(* IEC 61131-3 sources: generating_plc_code_with_llms/Code#1/ChatGPT_3.5/first run, 20 files *)

(* ---- 10.st ---- *)
//7.60s
//2
FUNCTION Sigmoid : REAL
VAR_INPUT
    x: REAL;  // Input value for the sigmoid function
END_VAR_INPUT
VAR_OUTPUT
    result: REAL;  // Result of the sigmoid function
END_VAR_OUTPUT

VAR
    exp_neg_x: REAL;
BEGIN
    exp_neg_x := EXP(-x);
    result := 1 / (1 + exp_neg_x);
END_FUNCTION

(* ---- 11.st ---- *)
//7.59s
//2
FUNCTION Sign : INT
VAR_INPUT
    value: REAL;  // Input value to determine the sign of
END_VAR_INPUT
VAR_OUTPUT
    sign: INT;    // Output sign value (-1, 0, or 1)
END_VAR_OUTPUT
BEGIN
    IF value < 0 THEN
        sign := -1;
    ELSIF value = 0 THEN
        sign := 0;
    ELSE
        sign := 1;
    END_IF
END_FUNCTION

(* ---- 12.st ---- *)
//8.05s
//2
FUNCTION HyperbolicSine : REAL
VAR_INPUT
    x: REAL;  // Input value for the hyperbolic sine function
END_VAR_INPUT
VAR_OUTPUT
    result: REAL;  // Result of the hyperbolic sine function
END_VAR_OUTPUT

VAR
    exp_x: REAL;
    exp_neg_x: REAL;
BEGIN
    exp_x := EXP(x);
    exp_neg_x := EXP(-x);
    result := (exp_x - exp_neg_x) / 2;
END_FUNCTION

(* ---- 14.st ---- *)
// 33.60s
// 3
FUNCTION FC1001 : BOOL
VAR_INPUT
    MeasuredValue: REAL;      // Measured value from the sensor
    SwitchingValue: REAL;     // Predetermined switching value
    HysteresisPercent: REAL;  // Switching hysteresis in percentage
END_VAR

VAR_OUTPUT
    Output: BOOL;  // Output indicating the state (ON or OFF)
END_VAR

VAR
    HysteresisValue: REAL;  // Calculated hysteresis value based on percentage
    SwitchOnThreshold: REAL; // Threshold for switching ON
    SwitchOffThreshold: REAL; // Threshold for switching OFF
END_VAR

METHOD CheckSwitching
    HysteresisValue := SwitchingValue * HysteresisPercent / 100.0;

    SwitchOnThreshold := SwitchingValue + HysteresisValue;
    SwitchOffThreshold := SwitchingValue - HysteresisValue;

    IF MeasuredValue > SwitchOnThreshold THEN
        Output := TRUE;  // Switch ON
    ELSIF MeasuredValue < SwitchOffThreshold THEN
        Output := FALSE; // Switch OFF
    END_IF
END_METHOD

END_FUNCTION

(* ---- 15.st ---- *)
// 25.63s
// 2
FUNCTION FC1002 : BOOL
VAR_INPUT
    E_A: BOOL;    // Switch for turning on/off the monitoring system
    Approach: BOOL;  // Signal from the ultrasonic sensor indicating an approach
END_VAR

VAR_OUTPUT
    P_HU: BOOL;  // Output for the acoustic warning signal
    P_AL: BOOL;  // Output for the alarm signal
    P1: BOOL;    // Output indicating the switched-on status
END_VAR

VAR
    Timer: TON := (PT := T#3s);  // Timer for tracking the duration of the approach
END_VAR

METHOD UltrasonicMonitoring
    IF E_A THEN
        P1 := TRUE;  // Monitoring system is switched on

        IF Approach THEN
            P_HU := TRUE;  // Acoustic warning signal is activated

            IF Timer(IN := TRUE).Q THEN
                // Approach duration exceeds 3 seconds, switch off warning and activate alarm
                P_HU := FALSE;
                P_AL := TRUE;
            END_IF
        ELSE
            // No approach, reset the timer and signals
            Timer(IN := FALSE);
            P_HU := FALSE;
            P_AL := FALSE;
        END_IF
    ELSE
        // Monitoring system is switched off, reset all signals
        P1 := FALSE;
        P_HU := FALSE;
        P_AL := FALSE;
        Timer(IN := FALSE);
    END_IF
END_METHOD

END_FUNCTION

(* ---- 18.st ---- *)
// 8.55s
// 2
FUNCTION FC1003
VAR_INPUT
    DigitalInput: INT;  // Digital input value (0 to 255)
    IN_MIN: INT;        // Lower limit of the original range
    IN_MAX: INT;        // Upper limit of the original range
    OUT_MIN: REAL;      // Lower limit of the output range
    OUT_MAX: REAL;      // Upper limit of the output range
END_VAR_INPUT

VAR_OUTPUT
    Temperature: REAL;  // Converted temperature value
END_VAR_OUTPUT

VAR
    M: REAL;            // Slope of the linear mapping
    B: REAL;            // Y-intercept of the linear mapping
END_VAR

// Calculate the slope and y-intercept for the linear mapping
M := (OUT_MAX - OUT_MIN) / (IN_MAX - IN_MIN);
B := OUT_MIN - M * IN_MIN;

// Perform the linear mapping to convert DigitalInput to Temperature
Temperature := M * DigitalInput + B;

END_FUNCTION

(* ---- 2.st ---- *)
//7.4s
//2
FUNCTION CalculateBinomialCoefficient : INT
VAR_INPUT
    n : INT;  // The total number of items (n)
    k : INT;  // The number of items to choose (k)
END_VAR_INPUT
VAR_OUTPUT
    result : INT;  // The binomial coefficient result
END_VAR_OUTPUT
VAR
    i : INT;
    numerator : INT := 1;
    denominator : INT := 1;
END_VAR

IF (k < 0) OR (k > n) THEN
    result := 0;  // Invalid input, return 0
ELSE
    FOR i := 1 TO k DO
        numerator := numerator * (n - i + 1);
        denominator := denominator * i;
    END_FOR

    result := numerator / denominator;
END_IF

END_FUNCTION

(* ---- 3.st ---- *)
//6.85s
//2
FUNCTION CalculateFibonacci : INT
VAR_INPUT
    n : INT;  // The position in the Fibonacci sequence (0-based)
END_VAR_INPUT
VAR_OUTPUT
    result : INT;  // The Fibonacci number at position 'n'
END_VAR_OUTPUT
VAR
    fibNMinus2 : INT := 0;  // Initial values for the first two Fibonacci numbers
    fibNMinus1 : INT := 1;
    fibN : INT;
    i : INT;
END_VAR

IF n = 0 THEN
    result := fibNMinus2;  // Special case for n = 0
ELSIF n = 1 THEN
    result := fibNMinus1;  // Special case for n = 1
ELSE
    FOR i := 2 TO n DO
        fibN := fibNMinus1 + fibNMinus2;
        fibNMinus2 := fibNMinus1;
        fibNMinus1 := fibN;
    END_FOR

    result := fibN;
END_IF

END_FUNCTION

(* ---- 19.st ---- *)
// 20.66s
// 3
FUNCTION_BLOCK FB1005
VAR_INPUT
    START: BOOL;      // Start the measurement (connected to sensor S1)
    THICKNESS: REAL;  // Input representing the thickness of the ceramic plate
    V_MAX: REAL;      // Maximum allowed thickness
    V_MIN: REAL;      // Minimum allowed thickness
END_VAR

VAR_OUTPUT
    M_MAX: REAL;      // Largest thickness recorded during the measurement
    M_MIN: REAL;      // Smallest thickness recorded during the measurement
    P1: BOOL;         // Output for the reject light
END_VAR

VAR
    D_MAX: BOOL;      // Flag indicating if the largest thickness is outside the specified range
    D_MIN: BOOL;      // Flag indicating if the smallest thickness is outside the specified range
    ThicknessStarted: BOOL;  // Flag indicating if the thickness measurement has started
    LastThickness: REAL;     // Last recorded thickness during the measurement
END_VAR

METHOD MeasureThickness
    IF START THEN
        // Start of a new measurement cycle
        M_MAX := THICKNESS;  // Initialize largest thickness
        M_MIN := THICKNESS;  // Initialize smallest thickness
        D_MAX := FALSE;      // Initialize flags
        D_MIN := FALSE;
        ThicknessStarted := TRUE;  // Set the flag to indicate the measurement has started
    END_IF

    IF ThicknessStarted THEN
        // During the measurement cycle
        IF THICKNESS > M_MAX THEN
            M_MAX := THICKNESS;  // Update largest thickness
        END_IF

        IF THICKNESS < M_MIN THEN
            M_MIN := THICKNESS;  // Update smallest thickness
        END_IF

        LastThickness := THICKNESS;  // Record the last thickness
    END_IF

    // After the measurement cycle
    IF NOT START AND ThicknessStarted THEN
        ThicknessStarted := FALSE;  // Reset the flag to indicate the end of the measurement
        D_MAX := M_MAX > V_MAX;     // Check if the largest thickness is outside the specified range
        D_MIN := M_MIN < V_MIN;     // Check if the smallest thickness is outside the specified range
    END_IF

    // Output the reject light signal
    P1 := D_MAX OR D_MIN;
END_METHOD

END_FUNCTION_BLOCK

(* ---- 21.st ---- *)
// 46.74s
// 2
FUNCTION_BLOCK BURNER
VAR_INPUT
    IN: BOOL;                  // Control input
    OVER_TEMP: BOOL;           // Boiler thermostat protection
    OIL_TEMP: BOOL;            // Signal indicating oil temperature reached
    MULTIPLE_IGNITION: BOOL;   // Enable multiple ignition after flame break
    STAGE2: BOOL;              // Activate second stage
END_VAR_INPUT

VAR_OUTPUT
    PRE_HEAT: BOOL;            // Fuel oil warming
    MOTOR: BOOL;               // Motor status
    FAN: BOOL;                 // Fan status
    IGNITION: BOOL;            // Ignition status
    OIL_VALVE: BOOL;           // Oil valve status
    STATUS: INT;               // Module status
    FAIL: BOOL;                // Failure indication
END_VAR_OUTPUT

VAR
    startTime: TIME;           // Start time for various stages
    locked: BOOL;              // Module lock status
END_VAR

METHOD StartBurner : BOOL
VAR
    elapsedTime: TIME;         // Elapsed time for various stages
BEGIN
    // Check if the module is locked
    IF locked THEN
        STATUS := 99;  // Module is locked
        RETURN FALSE;
    END_IF

    // Reset failure indication
    FAIL := FALSE;

    // Start sequence
    IF IN AND NOT OVER_TEMP THEN
        PRE_HEAT := TRUE;  // Fuel oil warming
        startTime := T;    // Record start time

        // Wait for OIL_TEMP signal within PRE_HEAT_TIME
        WHILE (T - startTime < PRE_HEAT_TIME) AND NOT OIL_TEMP DO
            // Check if OVER_TEMP signal received during waiting
            IF OVER_TEMP THEN
                STATUS := 9;  // Boiler overheating error
                RETURN FALSE;
            END_IF
        END_WHILE

        // Check if OIL_TEMP signal received within PRE_HEAT_TIME
        IF OIL_TEMP THEN
            MOTOR := TRUE;  // Start motor
            FAN := TRUE;    // Start fan

            // Wait for PRE_VENTILATION_TIME before ignition
            WHILE (T - startTime < PRE_VENTILATION_TIME) DO
                // Check if OVER_TEMP signal received during waiting
                IF OVER_TEMP THEN
                    STATUS := 9;  // Boiler overheating error
                    RETURN FALSE;
                END_IF
            END_WHILE

            IGNITION := TRUE;  // Turn on ignition

            // Wait for PPR_IGNITION_TIME before opening oil valve
            WHILE (T - startTime < PPR_IGNITION_TIME) DO
                // Check if OVER_TEMP signal received during waiting
                IF OVER_TEMP THEN
                    STATUS := 9;  // Boiler overheating error
                    RETURN FALSE;
                END_IF
            END_WHILE

            OIL_VALVE := TRUE;  // Open oil valve

            // Wait for POST_IGNITION_TIME after ignition
            WHILE (T - startTime < POST_IGNITION_TIME) DO
                // Check if OVER_TEMP signal received during waiting
                IF OVER_TEMP THEN
                    STATUS := 9;  // Boiler overheating error
                    RETURN FALSE;
                END_IF
            END_WHILE

            // Check if flame sensor is active during SAFETY_TIME
            IF FLAME_SENSOR_ACTIVE(DURATION := SAFETY_TIME) THEN
                STATUS := 4;  // Safety time error
                RETURN FALSE;
            END_IF

            // Successful operation in stage 1
            STATUS := 112;  // Burner runs on stage 1

            // If MULTIPLE_IGNITION is enabled and flame breaks off, restart ignition
            IF MULTIPLE_IGNITION AND FLAME_SENSOR_ACTIVE(DURATION := MULTIPLE_IGNITION_TIME) THEN
                IGNITION := TRUE;  // Restart ignition
            END_IF

            // Check if second stage is activated
            IF STAGE2 THEN
                // Wait for STAGE2_DELAY before activating second stage
                WHILE (T - startTime < STAGE2_DELAY) DO
                    // Check if OVER_TEMP signal received during waiting
                    IF OVER_TEMP THEN
                        STATUS := 9;  // Boiler overheating error
                        RETURN FALSE;
                    END_IF
                END_WHILE

                // Activate second stage
                STATUS := 113;  // Burner runs at stage 2
            END_IF

            // Burner operation completed successfully
            RETURN TRUE;
        ELSE
            // OIL_TEMP signal not received within PRE_HEAT_TIME
            STATUS := 1;  // Fuel oil warming not responded error
            FAIL := TRUE;
            RETURN FALSE;
        END_IF
    ELSE
        // IN or OVER_TEMP condition not met
        STATUS := 110;  // Wait for Start signal (Standby)
        RETURN FALSE;
    END_IF
END_METHOD

METHOD FLAME_SENSOR_ACTIVE : BOOL
VAR_INPUT
    DURATION: TIME;  // Duration to check flame sensor activity
END_VAR_INPUT

VAR
    startTime: TIME;  // Start time for flame sensor check
BEGIN
    startTime := T;

    WHILE (T - startTime < DURATION) DO
        // Check if flame sensor is active
        IF FLAME_SENSOR THEN
            STATUS := 2;  // Flame sensor active error
            FAIL := TRUE;
            RETURN TRUE;
        END_IF
    END_WHILE

    // Flame sensor not active within specified duration
    RETURN FALSE;
END_METHOD

METHOD Lockout : BOOL
VAR
    lockoutStartTime: TIME;  // Start time for lockout
BEGIN
    // Set the module to locked state
    locked := TRUE;

    // Start lockout timer
    lockoutStartTime := T;

    // Wait for LOCKOUT_TIME
    WHILE (T - lockoutStartTime < LOCKOUT_TIME) AND NOT RST DO
        // Check if OVER_TEMP signal received during waiting
        IF OVER_TEMP THEN
            STATUS := 9;  // Boiler overheating error
            FAIL := TRUE;
            RETURN FALSE;
        END_IF
    END_WHILE

    // Reset the module lock
    locked := FALSE;

    // Module is ready for operation again
    STATUS := 110;  // Wait for Start signal (Standby)

    // Return TRUE if RST signal received after LOCKOUT_TIME
    RETURN RST;
END_METHOD

END_FUNCTION_BLOCK

(* ---- 1.st ---- *)
// 5.73s
//3
PROGRAM AlarmControl
VAR
    xAlarm1: BOOL := FALSE;
    xAlarm2: BOOL := FALSE;
    xAllOn: BOOL := FALSE;
    xAllOff: BOOL := FALSE;
END_VAR

xAlarm1 := FALSE;  // Ensure alarms are initially turned off
xAlarm2 := FALSE;

IF xAllOn THEN
    xAlarm1 := TRUE;
    xAlarm2 := TRUE;
ELSIF xAllOff THEN
    xAlarm1 := FALSE;
    xAlarm2 := FALSE;
END_IF

// Rest of your program logic here

END_PROGRAM

(* ---- 13.st ---- *)
//12.85s
//2
PROGRAM NumberSearch
VAR
    NumberList: ARRAY[1..100] OF INT;  // Array of 100 random numbers
    NumberToFind: INT := 10;           // Number to search for
    NumberFound: BOOL := FALSE;        // Flag to indicate if the number is found
    i: INT := 1;                       // Loop counter
END_VAR

FOR i := 1 TO 100 DO
    NumberList[i] := RANDOM(1, 100);  // Replace with a function that generates random numbers

    IF NumberList[i] = NumberToFind THEN
        NumberFound := TRUE;  // The number 10 is found, abort the search
        EXIT;  // Exit the loop
    END_IF
END_FOR

IF NOT NumberFound THEN
    // The number 10 was not found in the list
    // Handle the case where the number does not exist
    // Your logic for this case goes here
END_IF

// Your program logic continues here

(* ---- 16.st ---- *)
//13.22s
//2
PROGRAM TrafficLightControl
VAR
    North_green: BOOL := FALSE;
    North_yellow: BOOL := FALSE;
    North_red: BOOL := FALSE;
    East_green: BOOL := FALSE;
    East_yellow: BOOL := FALSE;
    East_red: BOOL := FALSE;

    TrafficLightCycleTimer: TON := (PT := T#10000ms);
END_VAR

CASE TrafficLightCycleTimer.IN THEN
    0:  // Between 0ms and 5000ms
        North_green := TRUE;
        East_green := FALSE;
        East_red := TRUE;
    5000:  // After 5000ms, North light turns yellow
        North_green := FALSE;
        North_yellow := TRUE;
    5500:  // Between 5500ms and 9500ms
        North_yellow := FALSE;
        North_red := TRUE;
        East_green := TRUE;
        East_red := FALSE;
    9500:  // Between 9500ms and 10000ms
        East_green := FALSE;
        East_yellow := TRUE;
    10000:  // Reset the timer and the cycle
        TrafficLightCycleTimer(IN := FALSE, PT := T#10000ms);
        North_red := FALSE;
        East_yellow := FALSE;
        North_green := TRUE;
        East_red := TRUE;
END_CASE

TrafficLightCycleTimer(IN := TRUE);

(* ---- 17.st ---- *)
//10.91s
//4
PROGRAM WeatherStation
VAR
    TemperatureSensorValue: INT;   // Analog input value for temperature
    HumiditySensorValue: INT;      // Analog input value for humidity
    TemperatureText: STRING := ''; // Text representation of temperature status
    HumidityText: STRING := '';    // Text representation of humidity status
END_VAR

TemperatureSensorValue := YourTemperatureSensorFunction(); // Replace with your sensor reading
HumiditySensorValue := YourHumiditySensorFunction();       // Replace with your sensor reading

IF TemperatureSensorValue < 18 THEN
    TemperatureText := 'Cold';
ELSIF TemperatureSensorValue >= 18 AND TemperatureSensorValue <= 25 THEN
    IF HumiditySensorValue >= 40 AND HumiditySensorValue <= 75 THEN
        TemperatureText := 'Opt';
    ELSE
        TemperatureText := 'Temp. OK';
    END_IF;
ELSE
    TemperatureText := 'Hot';
END_IF

// Display the temperature status in the house
DISPLAY_IN_HOUSE(TemperatureText);

// Your program logic continues here

END_PROGRAM

(* ---- 20.st ---- *)
// 15.67s
// 3
PROGRAM InterlockProgram
VAR_INPUT
    I1: BOOL;  // Input to switch Q1
    I2: BOOL;  // Input to switch Q2
END_VAR

VAR_OUTPUT
    Q1: BOOL;  // Output Q1
    Q2: BOOL;  // Output Q2
END_VAR

VAR
    TimerQ1: TON := (PT := T#1s);  // Timer for Q1
    TimerQ2: TON := (PT := T#1s);  // Timer for Q2
    TL: TIME := T#500ms;           // Dead time between Q1 and Q2
    LastQ1State: BOOL := FALSE;    // Last state of Q1
    LastQ2State: BOOL := FALSE;    // Last state of Q2
END_VAR

METHOD InterlockLogic
    // Update timers
    TimerQ1(IN := I1);
    TimerQ2(IN := I2);

    // Determine the next state of Q1
    IF I1 AND NOT Q2 AND TimerQ2.Q THEN
        Q1 := TRUE;
        LastQ1State := TRUE;
    ELSIF NOT I1 THEN
        Q1 := FALSE;
        TimerQ1(IN := FALSE);  // Reset the timer if I1 is OFF
    END_IF

    // Determine the next state of Q2
    IF I2 AND NOT Q1 AND TimerQ1.Q THEN
        Q2 := TRUE;
        LastQ2State := TRUE;
    ELSIF NOT I2 THEN
        Q2 := FALSE;
        TimerQ2(IN := FALSE);  // Reset the timer if I2 is OFF
    END_IF

    // Check for mutual locking
    IF LastQ1State AND TimerQ2.ET < TL THEN
        Q1 := FALSE;
    END_IF

    IF LastQ2State AND TimerQ1.ET < TL THEN
        Q2 := FALSE;
    END_IF

    // Update last states
    LastQ1State := Q1;
    LastQ2State := Q2;
END_METHOD

END_PROGRAM

(* ---- 4.st ---- *)
//14.19s
//2
PROGRAM FillLevelMonitor
VAR
    AnalogValue: INT := 0;      // Analog value (0 - 32767)
    FillLevelPercentage: REAL;  // Fill level percentage (0 - 100%)
    LowLevel: BOOL := FALSE;    // Output for low fill level
    OkLevel: BOOL := FALSE;     // Output for ok fill level
    HighLevel: BOOL := FALSE;   // Output for high fill level
    WarningHorn: BOOL := FALSE; // Output for the warning horn
END_VAR

// Read the analog value (0 - 32767) from your sensor
AnalogValue := YourAnalogSensorFunction();  // Replace with your actual sensor reading

// Convert the analog value to a percentage (0 - 100%)
FillLevelPercentage := REAL(AnalogValue) / 327.67;

// Use the CASE instruction to categorize the fill level
CASE
    FillLevelPercentage < 1.0:
        WarningHorn := TRUE;
    FillLevelPercentage < 30.0:
        LowLevel := TRUE;
    FillLevelPercentage < 70.0:
        OkLevel := TRUE;
    ELSE
        HighLevel := TRUE;
END_CASE

// Reset other outputs to FALSE
IF WarningHorn = TRUE THEN
    LowLevel := FALSE;
    OkLevel := FALSE;
    HighLevel := FALSE;
ELSE
    WarningHorn := FALSE;
END_IF

// Your program logic continues here

END_PROGRAM

(* ---- 5.st ---- *)
//11.55s
//2
PROGRAM GateController
VAR
    Start_Loop: BOOL := TRUE;          // Start/Stop the loop
    One_Hour_Timer: TIME := T#1H;     // 1-hour timer
    Gate_Open: BOOL := FALSE;         // Gate status (initially closed)
    Auth_String: STRING := "my_defined_str";  // Authentication string
    App_Presence: BOOL := FALSE;       // App presence signal
    Car_Presence: BOOL := FALSE;       // Car presence signal
END_VAR

IF NOT Start_Loop THEN
    One_Hour_Timer := One_Hour_Timer - T#1S;  // Decrement the timer by 1 second
END_IF

IF One_Hour_Timer <= T#0S THEN
    IF Gate_Open THEN
        Gate_Open := FALSE;  // Close the gate as the timer has timed out
    END_IF
END_IF

IF (App_Presence OR Car_Presence) AND (Auth_String = "my_defined_str") THEN
    Gate_Open := TRUE;  // Open the gate when authorized and presence detected
    One_Hour_Timer := T#1H;  // Restart the timer
END_IF

// Your program logic continues here

END_PROGRAM

(* ---- 6.st ---- *)
//14.34s
// 2
PROGRAM CraneLiftControl
VAR
    doConvTop: BOOL := FALSE;        // Conveyor belt for top crates
    doConvBottom: BOOL := FALSE;     // Conveyor belt for bottom crates
    diConvTop: BOOL := FALSE;        // Light barrier for top conveyor
    diConvBottom: BOOL := FALSE;     // Light barrier for bottom conveyor
    doLiftTop: BOOL := FALSE;        // Lift to top position
    doLiftBottom: BOOL := FALSE;     // Lift to bottom position
    diLiftTop: BOOL := FALSE;        // Lift position at top
    diLiftBottom: BOOL := FALSE;     // Lift position at bottom
    doConvLift: BOOL := FALSE;       // Conveyor belt for lifting crate
    diBoxLift: BOOL := FALSE;        // Crate at lift sensor
    doLiftUnload: BOOL := FALSE;     // Lift to unloading position
    diLiftUnload: BOOL := FALSE;     // Lift position at unloading
END_VAR

VAR
    LiftRequested: BOOL := FALSE;    // Flag to indicate lift request
    BoxInLift: BOOL := FALSE;        // Flag to indicate a crate in the lift
END_VAR

CASE LiftRequested OF
    FALSE:
        IF diConvTop THEN
            doConvTop := FALSE;  // Stop top conveyor
            doLiftTop := TRUE;   // Move the lift to top position
            LiftRequested := TRUE;
        ELSIF diConvBottom THEN
            doConvBottom := FALSE;  // Stop bottom conveyor
            doLiftBottom := TRUE;   // Move the lift to bottom position
            LiftRequested := TRUE;
        END_IF;
    TRUE:
        IF diLiftTop AND NOT BoxInLift THEN
            doConvLift := TRUE;   // Activate the lift conveyor
        END_IF;
        IF diBoxLift THEN
            doConvLift := FALSE;  // Stop lift conveyor when crate is in lift
            BoxInLift := TRUE;
            doLiftUnload := TRUE;  // Move the lift to unloading position
        END_IF;
        IF diLiftUnload AND BoxInLift THEN
            doConvLift := TRUE;   // Activate lift conveyor to unload crate
        END_IF;
        IF NOT diBoxLift AND diLiftUnload THEN
            doConvLift := FALSE;  // Stop lift conveyor when crate is unloaded
            doLiftUnload := FALSE;  // Reset unloading position
            doConvTop := TRUE;  // Resume the conveyor
            doConvBottom := TRUE;
            doLiftTop := FALSE;  // Reset lift position
            doLiftBottom := FALSE;
            LiftRequested := FALSE;
            BoxInLift := FALSE;
        END_IF;
END_CASE

END_PROGRAM

(* ---- 7.st ---- *)
//9.39s
//2
PROGRAM CraneControl
VAR
    LoadReceptorValues: ARRAY[1..5] OF INT;  // Array to store load values for 5 receptors
    TotalLoad: INT := 0;  // Total load
    AverageLoad: INT := 0;  // Average load
    NumLoadReceptors: INT := 5;  // Number of load receptors (constant)
    AnalogInputRangeMin: INT := 0;  // Minimum value for analog inputs (constant)
    AnalogInputRangeMax: INT := 32767;  // Maximum value for analog inputs (constant)
END_VAR

FOR i := 1 TO NumLoadReceptors DO
    // Read analog values from load receptors (replace with actual readings)
    LoadReceptorValues[i] := ReadAnalogValue(i);  // Replace with your function

    // Ensure the values are within the specified range
    IF LoadReceptorValues[i] < AnalogInputRangeMin THEN
        LoadReceptorValues[i] := AnalogInputRangeMin;
    ELSIF LoadReceptorValues[i] > AnalogInputRangeMax THEN
        LoadReceptorValues[i] := AnalogInputRangeMax;
    END_IF

    TotalLoad := TotalLoad + LoadReceptorValues[i];  // Calculate total load
END_FOR

IF NumLoadReceptors > 0 THEN
    AverageLoad := TotalLoad / NumLoadReceptors;  // Calculate average load
ELSE
    AverageLoad := 0;  // Handle the case when there are no load receptors
END_IF

// Your program logic continues here

END_PROGRAM

(* ---- 9.st ---- *)
//7.57s
//4
PROGRAM LeapYearChecker
VAR
    YEAR: INT := 2024;  // Replace with the year you want to check
    IsLeapYear: BOOL := FALSE;
END_VAR

IF (YEAR MOD 4 = 0) AND ((YEAR MOD 100 <> 0) OR (YEAR MOD 400 = 0)) THEN
    IsLeapYear := TRUE;
ELSE
    IsLeapYear := FALSE;
END_IF

// Now you can use the IsLeapYear variable to determine if the year is a leap year or not

END_PROGRAM
